FUNCTION_BLOCK ActuatorsSimulation (* CAT Function Block Type *)
  (* Standard: 61499-2 *)
  (* Version 0.0, 7/3/2026, Schneider Electric, template *)
  PACKAGE SE.Nereda;
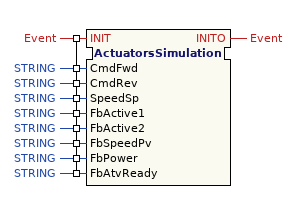
  EVENT_INPUT
    INIT WITH FbActive1, FbActive2, CmdFwd, SpeedSp, FbSpeedPv, CmdRev, FbPower, FbAtvReady; (* Initializes the symbolic link data source FB with N (1 <= N <= 16) variables *)
  END_EVENT
  EVENT_OUTPUT
    INITO; (* Initialization confirm *)
  END_EVENT
  VAR_INPUT
    CmdFwd : STRING;
    CmdRev : STRING;
    SpeedSp : STRING;
    FbActive1 : STRING;
    FbActive2 : STRING;
    FbSpeedPv : STRING;
    FbPower : STRING;
    FbAtvReady : STRING;
  END_VAR
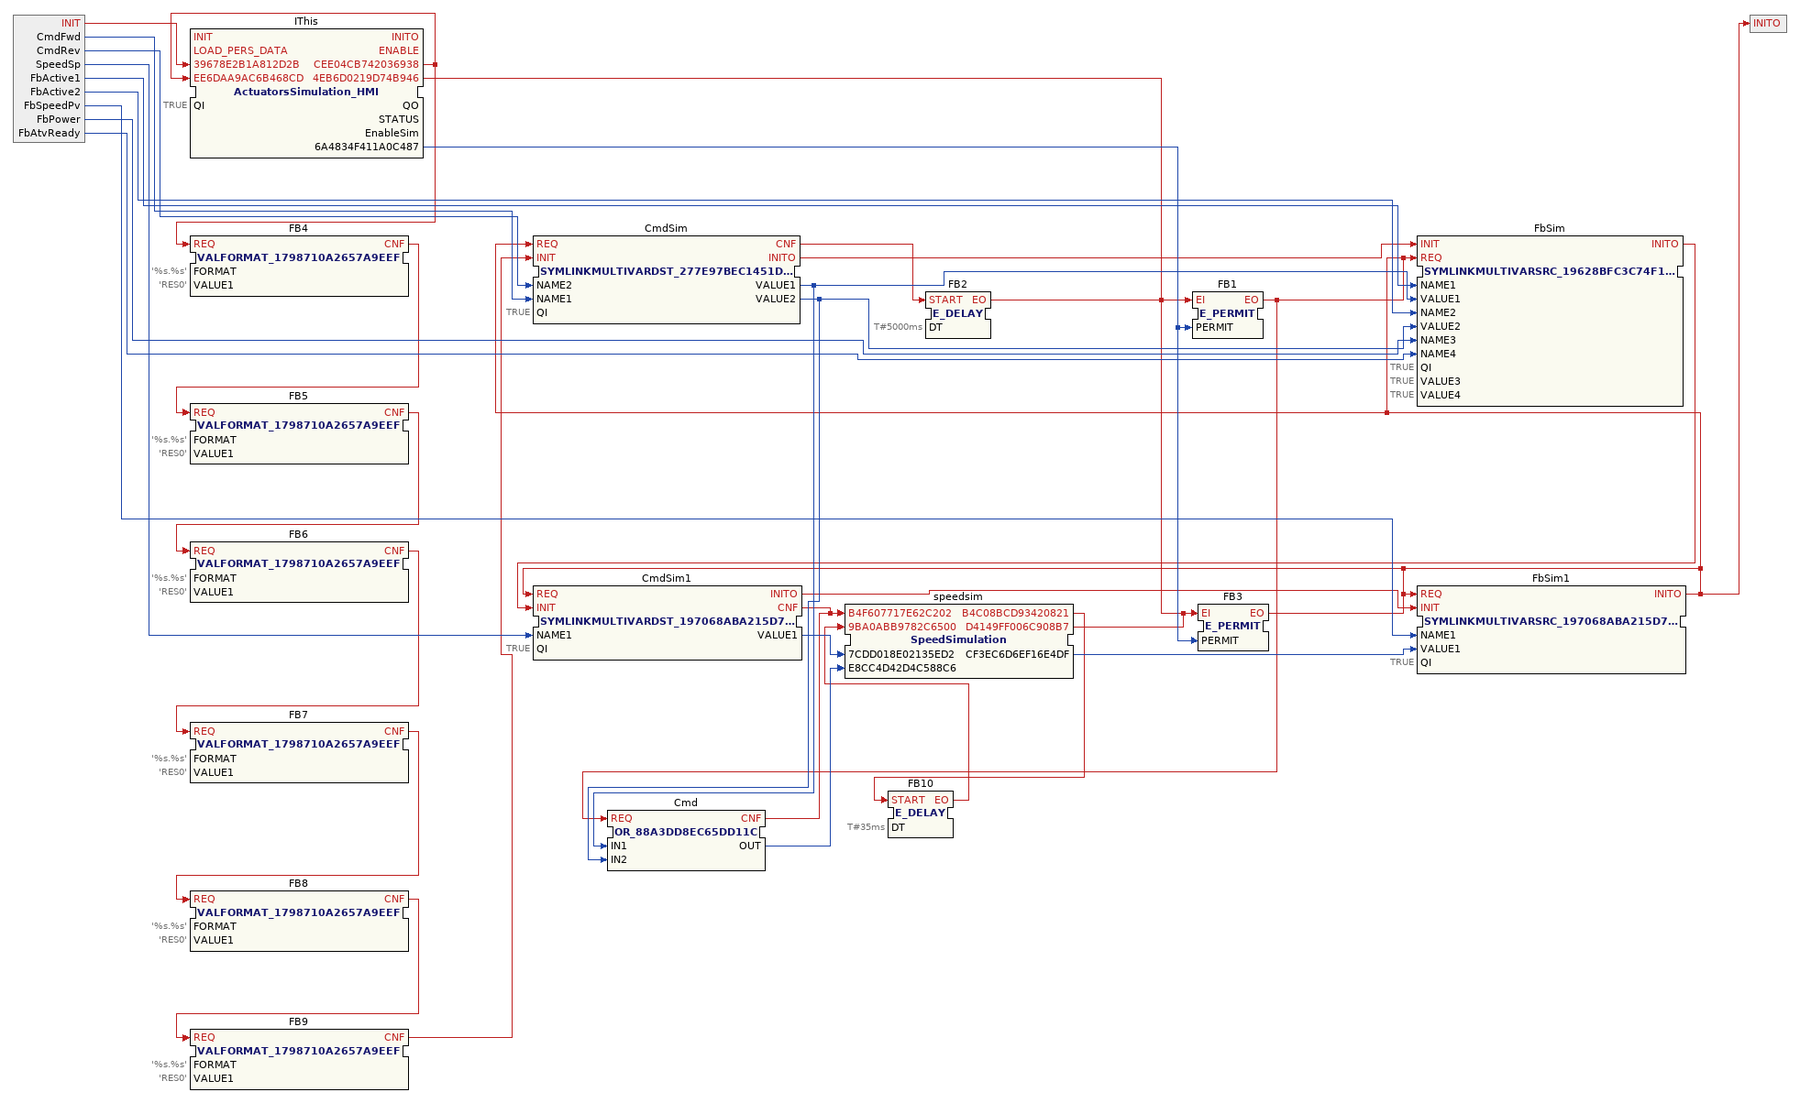
  FBS
    FbSim : SYMLINKMULTIVARSRC_19628BFC3C74F1AB1(QI := TRUE, VALUE3 := TRUE, VALUE4 := TRUE); {SET_ATTRIBUTE(Configuration.GenericFBType.InterfaceParams, Runtime.System#I:=4;VALUE${I$}:BOOL,BOOL,BOOL,BOOL)}
    CmdSim : SYMLINKMULTIVARDST_277E97BEC1451D2C(QI := TRUE); {SET_ATTRIBUTE(Configuration.GenericFBType.InterfaceParams, Runtime.System#I:=2;VALUE${I$}:BOOL,BOOL)}
    FB2 : E_DELAY(DT := T#5000ms);
    FbSim1 : SYMLINKMULTIVARSRC_197068ABA215D7EBA(QI := TRUE); {SET_ATTRIBUTE(Configuration.GenericFBType.InterfaceParams, Runtime.System#I:=1;VALUE${I$}:REAL)}
    CmdSim1 : SYMLINKMULTIVARDST_197068ABA215D7EBA(QI := TRUE); {SET_ATTRIBUTE(Configuration.GenericFBType.InterfaceParams, Runtime.System#I:=1;VALUE${I$}:REAL)}
    FB1 : E_PERMIT;
    FB3 : E_PERMIT;
    FB4 : VALFORMAT_1798710A2657A9EEF(FORMAT := '%s.%s', VALUE1 := 'RES0'); {SET_ATTRIBUTE(Configuration.GenericFBType.InterfaceParams, Runtime.Standard#I:=2;VALUE${I$}:STRING,STRING)}
    FB5 : VALFORMAT_1798710A2657A9EEF(FORMAT := '%s.%s', VALUE1 := 'RES0'); {SET_ATTRIBUTE(Configuration.GenericFBType.InterfaceParams, Runtime.Standard#I:=2;VALUE${I$}:STRING,STRING)}
    FB6 : VALFORMAT_1798710A2657A9EEF(FORMAT := '%s.%s', VALUE1 := 'RES0'); {SET_ATTRIBUTE(Configuration.GenericFBType.InterfaceParams, Runtime.Standard#I:=2;VALUE${I$}:STRING,STRING)}
    FB7 : VALFORMAT_1798710A2657A9EEF(FORMAT := '%s.%s', VALUE1 := 'RES0'); {SET_ATTRIBUTE(Configuration.GenericFBType.InterfaceParams, Runtime.Standard#I:=2;VALUE${I$}:STRING,STRING)}
    FB8 : VALFORMAT_1798710A2657A9EEF(FORMAT := '%s.%s', VALUE1 := 'RES0'); {SET_ATTRIBUTE(Configuration.GenericFBType.InterfaceParams, Runtime.Standard#I:=2;VALUE${I$}:STRING,STRING)}
    FB9 : VALFORMAT_1798710A2657A9EEF(FORMAT := '%s.%s', VALUE1 := 'RES0'); {SET_ATTRIBUTE(Configuration.GenericFBType.InterfaceParams, Runtime.Standard#I:=2;VALUE${I$}:STRING,STRING)}
    speedsim : SpeedSimulation;
    Cmd : OR_88A3DD8EC65DD11C; {SET_ATTRIBUTE(Configuration.GenericFBType.InterfaceParams, Runtime.Standard#CNT:=2;OUT:BOOL)}
    FB10 : E_DELAY(DT := T#35ms);
    IThis : ActuatorsSimulation_HMI(QI := TRUE);
  END_FBS
  EVENT_CONNECTIONS
    FbSim1.INITO TO INITO;
    FB2.EO TO FB1.EI;
    FB3.EO TO FbSim1.REQ;
    CmdSim.CNF TO FB2.START;
    INIT TO IThis.39678E2B1A812D2B;
    CmdSim.INITO TO FbSim.INIT;
    FB1.EO TO FbSim.REQ;
    CmdSim1.INITO TO FbSim1.INIT;
    FbSim1.INITO TO FbSim1.REQ;
    FbSim1.INITO TO CmdSim1.REQ;
    FbSim1.INITO TO CmdSim.REQ;
    FB4.CNF TO FB5.REQ;
    FB5.CNF TO FB6.REQ;
    FB7.CNF TO FB8.REQ;
    FB8.CNF TO FB9.REQ;
    FB6.CNF TO FB7.REQ;
    FB9.CNF TO CmdSim.INIT;
    FB1.EO TO Cmd.REQ;
    FbSim1.INITO TO FbSim.REQ;
    FbSim.INITO TO CmdSim1.INIT;
    IThis.CEE04CB742036938 TO FB4.REQ;
    IThis.CEE04CB742036938 TO IThis.EE6DAA9AC6B468CD;
    IThis.4EB6D0219D74B946 TO FB1.EI;
    IThis.4EB6D0219D74B946 TO FB3.EI;
    CmdSim1.CNF TO speedsim.B4F607717E62C202;
    Cmd.CNF TO speedsim.B4F607717E62C202;
    FB10.EO TO speedsim.9BA0ABB9782C6500;
    speedsim.B4C08BCD93420821 TO FB10.START;
    speedsim.D4149FF006C908B7 TO FB3.EI;
  END_CONNECTIONS
  DATA_CONNECTIONS
    IThis.6A4834F411A0C487 TO FB1.PERMIT;
    IThis.6A4834F411A0C487 TO FB3.PERMIT;
    CmdRev TO CmdSim.NAME2;
    SpeedSp TO CmdSim1.NAME1;
    CmdFwd TO CmdSim.NAME1;
    FbSpeedPv TO FbSim1.NAME1;
    CmdSim.VALUE1 TO Cmd.IN1;
    CmdSim.VALUE2 TO Cmd.IN2;
    FbActive1 TO FbSim.NAME1;
    CmdSim.VALUE1 TO FbSim.VALUE1;
    FbActive2 TO FbSim.NAME2;
    CmdSim.VALUE2 TO FbSim.VALUE2;
    FbPower TO FbSim.NAME3;
    FbAtvReady TO FbSim.NAME4;
    CmdSim1.VALUE1 TO speedsim.7CDD018E02135ED2;
    Cmd.OUT TO speedsim.E8CC4D42D4C588C6;
    speedsim.CF3EC6D6EF16E4DF TO FbSim1.VALUE1;
  END_CONNECTIONS
END_FUNCTION_BLOCK
